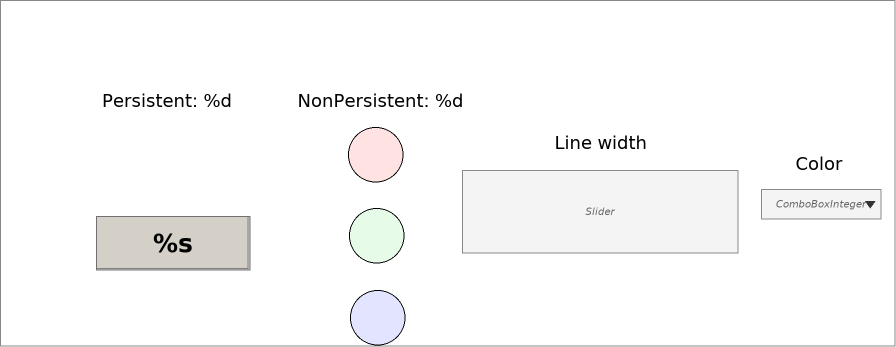
VISUALIZATION VisuAmpel  // 896x347
    Button (96,216 154x54), "%s", text variable: MAIN.btnText
        OnMouseDown: execute { MAIN.btnSwitch:=true; }
        OnMouseUp: execute { MAIN.btnSwitch:=FALSE; }
    Ellipse (348,127 55x55), colour toggle: MAIN.bLightR
        p1271844420: MAIN.iWidth
    Slider (462,170 276x83), variable: MAIN.iIntensity, invisible if: not MAIN.bLight, scale 0..8
    Rectangle (62,78 210x46), "Persistent: %d", text variable: MAIN.iCounterP
    Rectangle (273,78 215x46), "NonPersistent: %d", text variable: MAIN.iCounter
    Ellipse (349,208 55x55), colour toggle: MAIN.bLightG
        p1271844420: MAIN.iWidth
    Ellipse (350,290 55x55), colour toggle: MAIN.bLightB
        p1271844420: MAIN.iWidth
    ComboBoxInteger (761,189 120x30), tooltip "Color", variable: MAIN.iColor, invisible if: not MAIN.bLight, text list: 'Colors'
    Label (526,128 150x30), "Line width", invisible if: not MAIN.bLight
    Label (744,149 150x30), "Color", invisible if: not MAIN.bLight
END_VISUALIZATION

(* stored: Version 1.1.0.1, ProductVersion 3.1.4018.10
   Visu VisuAmpel: Id {64c0b840-b94a-4534-b255-25db3e63ffa3} *)
